ABB RAPID module: P701.mod

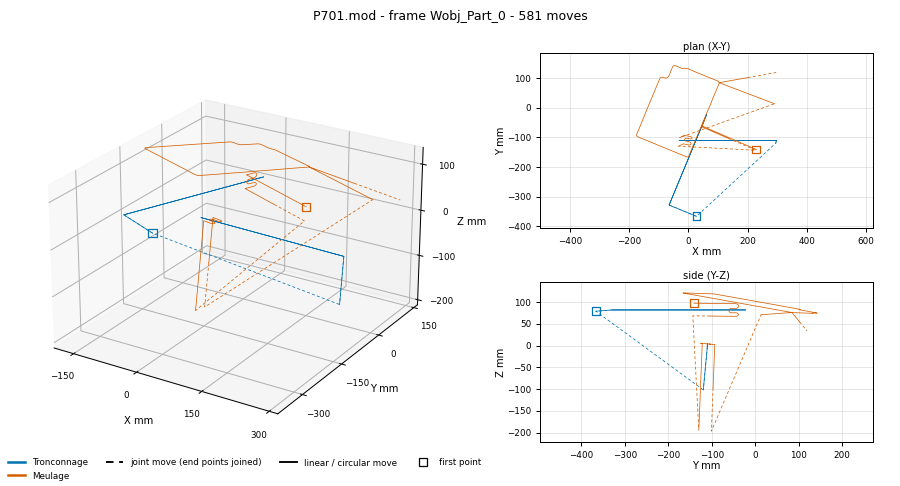
[picture p0: tool path of P701.mod in frame Wobj_Part_0, 581 of 591 moves have a stored position in this frame; points joined in program order, loops and branches not executed]
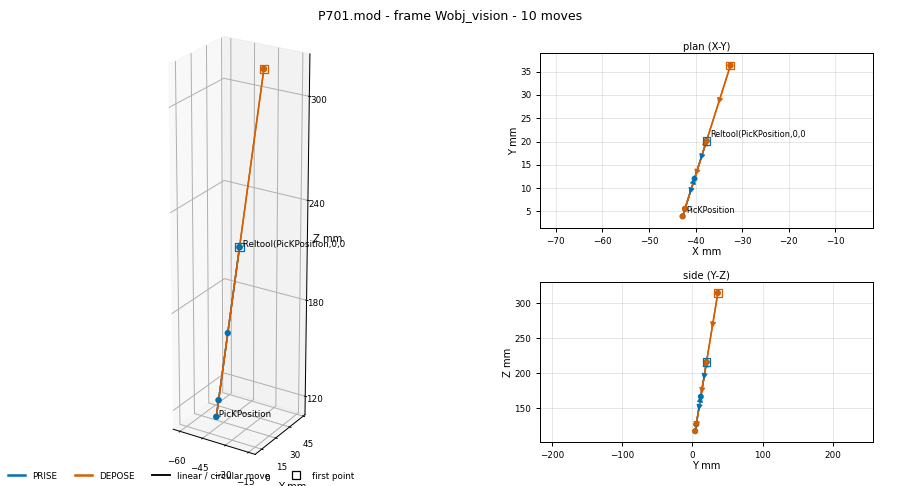
[picture p1: tool path of P701.mod in frame Wobj_vision, 10 of 591 moves have a stored position in this frame; points joined in program order, loops and branches not executed]
MODULE P701

    ! Nom         :P701
    ! Description :
    ! Créé le     :25/05/2023 17:26:44

    LOCAL CONST SPEEDDATA VitesseLente :=[10,500,0,0];
	LOCAL CONST SPEEDDATA VitesseRapide :=[30,500,0,0];
    !
    !Point de prise
    LOCAL PERS Robtarget PicKPosition := [[-42.7800235007069,3.94855808241573,117.453387874521],[0.0538335534292102,0.833835492186198,0.545408190576733,-0.0659562441896086],[0,0,0,0],[8.999999E+09,8.999999E+09,8.999999E+09,8.999999E+09,8.999999E+09,8.999999E+09]];
	LOCAL PERS Pose Ref := [[0,0,0],[1,0,0,0]];
    !
    !Declaration des points de meulage

    !Tr_meulage_motif_1 : Meulage d'un motif
    LOCAL CONST Robtarget Tr_meulage_motif_1_0 := [[45.67339453125,-61.43734375,96.697234375],[0.589642666457992,-0.592820387806933,-0.388910456451629,0.386825762527953],[0,0,0,0],[8.999999E+09,8.999999E+09,8.999999E+09,8.999999E+09,8.999999E+09,8.999999E+09]];
    LOCAL CONST Robtarget Tr_meulage_motif_1_1 := [[46.0576171875,-60.5141015625,96.6973125],[0.589642666457992,-0.592820387806933,-0.388910456451629,0.386825762527953],[0,0,0,0],[8.999999E+09,8.999999E+09,8.999999E+09,8.999999E+09,8.999999E+09,8.999999E+09]];
    LOCAL CONST Robtarget Tr_meulage_motif_1_2 := [[46.44183984375,-59.590859375,96.6973828125],[0.589642666457992,-0.592820387806933,-0.388910456451629,0.386825762527953],[0,0,0,0],[8.999999E+09,8.999999E+09,8.999999E+09,8.999999E+09,8.999999E+09,8.999999E+09]];
    LOCAL CONST Robtarget Tr_meulage_motif_1_3 := [[46.8260625,-58.66762109375,96.6974609375],[0.589642666457992,-0.592820387806933,-0.388910456451629,0.386825762527953],[0,0,0,0],[8.999999E+09,8.999999E+09,8.999999E+09,8.999999E+09,8.999999E+09,8.999999E+09]];
    LOCAL CONST Robtarget Tr_meulage_motif_1_4 := [[47.21028125,-57.74437890625,96.6975390625],[0.589642666457992,-0.592820387806933,-0.388910456451629,0.386825762527953],[0,0,0,0],[8.999999E+09,8.999999E+09,8.999999E+09,8.999999E+09,8.999999E+09,8.999999E+09]];
    LOCAL CONST Robtarget Tr_meulage_motif_1_5 := [[47.59450390625,-56.82113671875,96.697609375],[0.589642666457992,-0.592820387806933,-0.388910456451629,0.386825762527953],[0,0,0,0],[8.999999E+09,8.999999E+09,8.999999E+09,8.999999E+09,8.999999E+09,8.999999E+09]];
    LOCAL CONST Robtarget Tr_meulage_motif_1_6 := [[47.9787265625,-55.8978984375,96.6976875],[0.589642666457992,-0.592820387806933,-0.388910456451629,0.386825762527953],[0,0,0,0],[8.999999E+09,8.999999E+09,8.999999E+09,8.999999E+09,8.999999E+09,8.999999E+09]];
    LOCAL CONST Robtarget Tr_meulage_motif_1_7 := [[48.36294921875,-54.97465625,96.697765625],[0.589642666457992,-0.592820387806933,-0.388910456451629,0.386825762527953],[0,0,0,0],[8.999999E+09,8.999999E+09,8.999999E+09,8.999999E+09,8.999999E+09,8.999999E+09]];
    LOCAL CONST Robtarget Tr_meulage_motif_1_8 := [[48.74716796875,-54.0514140625,96.69784375],[0.589642666457992,-0.592820387806933,-0.388910456451629,0.386825762527953],[0,0,0,0],[8.999999E+09,8.999999E+09,8.999999E+09,8.999999E+09,8.999999E+09,8.999999E+09]];
    LOCAL CONST Robtarget Tr_meulage_motif_1_9 := [[49.131390625,-53.12817578125,96.6979140625],[0.589642666457992,-0.592820387806933,-0.388910456451629,0.386825762527953],[0,0,0,0],[8.999999E+09,8.999999E+09,8.999999E+09,8.999999E+09,8.999999E+09,8.999999E+09]];
    LOCAL CONST Robtarget Tr_meulage_motif_1_10 := [[49.51561328125,-52.20493359375,96.6979921875],[0.589642666457992,-0.592820387806933,-0.388910456451629,0.386825762527953],[0,0,0,0],[8.999999E+09,8.999999E+09,8.999999E+09,8.999999E+09,8.999999E+09,8.999999E+09]];
    LOCAL CONST Robtarget Tr_meulage_motif_1_11 := [[49.8998359375,-51.28169140625,96.6980703125],[0.589642666457992,-0.592820387806933,-0.388910456451629,0.386825762527953],[0,0,0,0],[8.999999E+09,8.999999E+09,8.999999E+09,8.999999E+09,8.999999E+09,8.999999E+09]];
    LOCAL CONST Robtarget Tr_meulage_motif_1_12 := [[50.28405859375,-50.358453125,96.698140625],[0.589642666457992,-0.592820387806933,-0.388910456451629,0.386825762527953],[0,0,0,0],[8.999999E+09,8.999999E+09,8.999999E+09,8.999999E+09,8.999999E+09,8.999999E+09]];
    LOCAL CONST Robtarget Tr_meulage_motif_1_13 := [[50.66827734375,-49.4352109375,96.69821875],[0.589642666457992,-0.592820387806933,-0.388910456451629,0.386825762527953],[0,0,0,0],[8.999999E+09,8.999999E+09,8.999999E+09,8.999999E+09,8.999999E+09,8.999999E+09]];
    LOCAL CONST Robtarget Tr_meulage_motif_1_14 := [[51.0525,-48.51196875,96.698296875],[0.589642666457992,-0.592820387806933,-0.388910456451629,0.386825762527953],[0,0,0,0],[8.999999E+09,8.999999E+09,8.999999E+09,8.999999E+09,8.999999E+09,8.999999E+09]];
    LOCAL CONST Robtarget Tr_meulage_motif_1_15 := [[51.43672265625,-47.58873046875,96.698375],[0.589642666457992,-0.592820387806933,-0.388910456451629,0.386825762527953],[0,0,0,0],[8.999999E+09,8.999999E+09,8.999999E+09,8.999999E+09,8.999999E+09,8.999999E+09]];
    LOCAL CONST Robtarget Tr_meulage_motif_1_16 := [[51.8209453125,-46.66548828125,96.6984453125],[0.589642666457992,-0.592820387806933,-0.388910456451629,0.386825762527953],[0,0,0,0],[8.999999E+09,8.999999E+09,8.999999E+09,8.999999E+09,8.999999E+09,8.999999E+09]];
    LOCAL CONST Robtarget Tr_meulage_motif_1_17 := [[52.2051640625,-45.74225,96.6985234375],[0.589642666457992,-0.592820387806933,-0.388910456451629,0.386825762527953],[0,0,0,0],[8.999999E+09,8.999999E+09,8.999999E+09,8.999999E+09,8.999999E+09,8.999999E+09]];
    LOCAL CONST Robtarget Tr_meulage_motif_1_18 := [[52.58938671875,-44.8190078125,96.6986015625],[0.589642666457992,-0.592820387806933,-0.388910456451629,0.386825762527953],[0,0,0,0],[8.999999E+09,8.999999E+09,8.999999E+09,8.999999E+09,8.999999E+09,8.999999E+09]];
    LOCAL CONST Robtarget Tr_meulage_motif_1_19 := [[52.96788671875,-43.9014296875,96.588125],[0.589642666457992,-0.592820387806933,-0.388910456451629,0.386825762527953],[0,0,0,0],[8.999999E+09,8.999999E+09,8.999999E+09,8.999999E+09,8.999999E+09,8.999999E+09]];
    LOCAL CONST Robtarget Tr_meulage_motif_1_20 := [[53.326078125,-43.0252890625,96.37709375],[0.589642666457992,-0.592820387806933,-0.388910456451629,0.386825762527953],[0,0,0,0],[8.999999E+09,8.999999E+09,8.999999E+09,8.999999E+09,8.999999E+09,8.999999E+09]];
    LOCAL CONST Robtarget Tr_meulage_motif_1_21 := [[53.6466640625,-42.2350703125,96.105421875],[0.589642666457992,-0.592820387806933,-0.388910456451629,0.386825762527953],[0,0,0,0],[8.999999E+09,8.999999E+09,8.999999E+09,8.999999E+09,8.999999E+09,8.999999E+09]];
    LOCAL CONST Robtarget Tr_meulage_motif_1_22 := [[53.92765625,-41.53969921875,95.8296484375],[0.589642666457992,-0.592820387806933,-0.388910456451629,0.386825762527953],[0,0,0,0],[8.999999E+09,8.999999E+09,8.999999E+09,8.999999E+09,8.999999E+09,8.999999E+09]];
    LOCAL CONST Robtarget Tr_meulage_motif_1_23 := [[54.3347421875,-40.51645703125,95.2138515625],[0.589642666457992,-0.592820387806933,-0.388910456451629,0.386825762527953],[0,0,0,0],[8.999999E+09,8.999999E+09,8.999999E+09,8.999999E+09,8.999999E+09,8.999999E+09]];
    LOCAL CONST Robtarget Tr_meulage_motif_1_24 := [[54.70616796875,-39.5619609375,94.366609375],[0.589642666457992,-0.592820387806933,-0.388910456451629,0.386825762527953],[0,0,0,0],[8.999999E+09,8.999999E+09,8.999999E+09,8.999999E+09,8.999999E+09,8.999999E+09]];
    LOCAL CONST Robtarget Tr_meulage_motif_1_25 := [[55.0053203125,-38.7682421875,93.343203125],[0.589642666457992,-0.592820387806933,-0.388910456451629,0.386825762527953],[0,0,0,0],[8.999999E+09,8.999999E+09,8.999999E+09,8.999999E+09,8.999999E+09,8.999999E+09]];
    LOCAL CONST Robtarget Tr_meulage_motif_1_26 := [[55.16394921875,-38.30542578125,92.2274921875],[0.589642666457992,-0.592820387806933,-0.388910456451629,0.386825762527953],[0,0,0,0],[8.999999E+09,8.999999E+09,8.999999E+09,8.999999E+09,8.999999E+09,8.999999E+09]];
    LOCAL CONST Robtarget Tr_meulage_motif_1_27 := [[55.1563125,-38.272875,91.531796875],[0.589642666457992,-0.592820387806933,-0.388910456451629,0.386825762527953],[0,0,0,0],[8.999999E+09,8.999999E+09,8.999999E+09,8.999999E+09,8.999999E+09,8.999999E+09]];
    LOCAL CONST Robtarget Tr_meulage_motif_1_28 := [[55.139171875,-38.26569140625,90.8708125],[0.589642666457992,-0.592820387806933,-0.388910456451629,0.386825762527953],[0,0,0,0],[8.999999E+09,8.999999E+09,8.999999E+09,8.999999E+09,8.999999E+09,8.999999E+09]];
    LOCAL CONST Robtarget Tr_meulage_motif_1_29 := [[55.10095703125,-38.30916796875,90.2099765625],[0.589642666457992,-0.592820387806933,-0.388910456451629,0.386825762527953],[0,0,0,0],[8.999999E+09,8.999999E+09,8.999999E+09,8.999999E+09,8.999999E+09,8.999999E+09]];
    LOCAL CONST Robtarget Tr_meulage_motif_1_30 := [[54.88097265625,-38.75716796875,89.108625],[0.589642666457992,-0.592820387806933,-0.388910456451629,0.386825762527953],[0,0,0,0],[8.999999E+09,8.999999E+09,8.999999E+09,8.999999E+09,8.999999E+09,8.999999E+09]];
    LOCAL CONST Robtarget Tr_meulage_motif_1_31 := [[54.52575,-39.5371015625,88.102328125],[0.589642666457992,-0.592820387806933,-0.388910456451629,0.386825762527953],[0,0,0,0],[8.999999E+09,8.999999E+09,8.999999E+09,8.999999E+09,8.999999E+09,8.999999E+09]];
    LOCAL CONST Robtarget Tr_meulage_motif_1_32 := [[54.1110546875,-40.47294140625,87.273703125],[0.589642666457992,-0.592820387806933,-0.388910456451629,0.386825762527953],[0,0,0,0],[8.999999E+09,8.999999E+09,8.999999E+09,8.999999E+09,8.999999E+09,8.999999E+09]];
    LOCAL CONST Robtarget Tr_meulage_motif_1_33 := [[53.83680078125,-41.10299609375,86.8780625],[0.589642666457992,-0.592820387806933,-0.388910456451629,0.386825762527953],[0,0,0,0],[8.999999E+09,8.999999E+09,8.999999E+09,8.999999E+09,8.999999E+09,8.999999E+09]];
    LOCAL CONST Robtarget Tr_meulage_motif_1_34 := [[53.37917578125,-42.166953125,86.3906328125],[0.589642666457992,-0.592820387806933,-0.388910456451629,0.386825762527953],[0,0,0,0],[8.999999E+09,8.999999E+09,8.999999E+09,8.999999E+09,8.999999E+09,8.999999E+09]];
    LOCAL CONST Robtarget Tr_meulage_motif_1_35 := [[53.04765234375,-42.94425,86.126578125],[0.589642666457992,-0.592820387806933,-0.388910456451629,0.386825762527953],[0,0,0,0],[8.999999E+09,8.999999E+09,8.999999E+09,8.999999E+09,8.999999E+09,8.999999E+09]];
    LOCAL CONST Robtarget Tr_meulage_motif_1_36 := [[52.6842578125,-43.80248828125,85.9221171875],[0.589642666457992,-0.592820387806933,-0.388910456451629,0.386825762527953],[0,0,0,0],[8.999999E+09,8.999999E+09,8.999999E+09,8.999999E+09,8.999999E+09,8.999999E+09]];
    LOCAL CONST Robtarget Tr_meulage_motif_1_37 := [[52.30430859375,-44.70752734375,85.8134921875],[0.589642666457992,-0.592820387806933,-0.388910456451629,0.386825762527953],[0,0,0,0],[8.999999E+09,8.999999E+09,8.999999E+09,8.999999E+09,8.999999E+09,8.999999E+09]];
    LOCAL CONST Robtarget Tr_meulage_motif_1_38 := [[51.920078125,-45.62269921875,85.7028671875],[0.589642666457992,-0.592820387806933,-0.388910456451629,0.386825762527953],[0,0,0,0],[8.999999E+09,8.999999E+09,8.999999E+09,8.999999E+09,8.999999E+09,8.999999E+09]];
    LOCAL CONST Robtarget Tr_meulage_motif_1_39 := [[51.53585546875,-46.54594140625,85.702796875],[0.589642666457992,-0.592820387806933,-0.388910456451629,0.386825762527953],[0,0,0,0],[8.999999E+09,8.999999E+09,8.999999E+09,8.999999E+09,8.999999E+09,8.999999E+09]];
    LOCAL CONST Robtarget Tr_meulage_motif_1_40 := [[51.1516328125,-47.4691796875,85.70271875],[0.589642666457992,-0.592820387806933,-0.388910456451629,0.386825762527953],[0,0,0,0],[8.999999E+09,8.999999E+09,8.999999E+09,8.999999E+09,8.999999E+09,8.999999E+09]];
    LOCAL CONST Robtarget Tr_meulage_motif_1_41 := [[50.76741015625,-48.392421875,85.702640625],[0.589642666457992,-0.592820387806933,-0.388910456451629,0.386825762527953],[0,0,0,0],[8.999999E+09,8.999999E+09,8.999999E+09,8.999999E+09,8.999999E+09,8.999999E+09]];
    LOCAL CONST Robtarget Tr_meulage_motif_1_42 := [[50.38319140625,-49.3156640625,85.7025625],[0.589642666457992,-0.592820387806933,-0.388910456451629,0.386825762527953],[0,0,0,0],[8.999999E+09,8.999999E+09,8.999999E+09,8.999999E+09,8.999999E+09,8.999999E+09]];
    LOCAL CONST Robtarget Tr_meulage_motif_1_43 := [[49.99896875,-50.23890234375,85.7024921875],[0.589642666457992,-0.592820387806933,-0.388910456451629,0.386825762527953],[0,0,0,0],[8.999999E+09,8.999999E+09,8.999999E+09,8.999999E+09,8.999999E+09,8.999999E+09]];
    LOCAL CONST Robtarget Tr_meulage_motif_1_44 := [[49.61474609375,-51.16214453125,85.7024140625],[0.589642666457992,-0.592820387806933,-0.388910456451629,0.386825762527953],[0,0,0,0],[8.999999E+09,8.999999E+09,8.999999E+09,8.999999E+09,8.999999E+09,8.999999E+09]];
    LOCAL CONST Robtarget Tr_meulage_motif_1_45 := [[49.2305234375,-52.08538671875,85.7023359375],[0.589642666457992,-0.592820387806933,-0.388910456451629,0.386825762527953],[0,0,0,0],[8.999999E+09,8.999999E+09,8.999999E+09,8.999999E+09,8.999999E+09,8.999999E+09]];
    LOCAL CONST Robtarget Tr_meulage_motif_1_46 := [[48.84630078125,-53.008625,85.7022578125],[0.589642666457992,-0.592820387806933,-0.388910456451629,0.386825762527953],[0,0,0,0],[8.999999E+09,8.999999E+09,8.999999E+09,8.999999E+09,8.999999E+09,8.999999E+09]];
    LOCAL CONST Robtarget Tr_meulage_motif_1_47 := [[48.46208203125,-53.9318671875,85.7021875],[0.589642666457992,-0.592820387806933,-0.388910456451629,0.386825762527953],[0,0,0,0],[8.999999E+09,8.999999E+09,8.999999E+09,8.999999E+09,8.999999E+09,8.999999E+09]];
    LOCAL CONST Robtarget Tr_meulage_motif_1_48 := [[48.077859375,-54.855109375,85.702109375],[0.589642666457992,-0.592820387806933,-0.388910456451629,0.386825762527953],[0,0,0,0],[8.999999E+09,8.999999E+09,8.999999E+09,8.999999E+09,8.999999E+09,8.999999E+09]];
    LOCAL CONST Robtarget Tr_meulage_motif_1_49 := [[47.69362890625,-55.77028125,85.591484375],[0.589642666457992,-0.592820387806933,-0.388910456451629,0.386825762527953],[0,0,0,0],[8.999999E+09,8.999999E+09,8.999999E+09,8.999999E+09,8.999999E+09,8.999999E+09]];
    LOCAL CONST Robtarget Tr_meulage_motif_1_50 := [[47.32448828125,-56.64183203125,85.3803046875],[0.589642666457992,-0.592820387806933,-0.388910456451629,0.386825762527953],[0,0,0,0],[8.999999E+09,8.999999E+09,8.999999E+09,8.999999E+09,8.999999E+09,8.999999E+09]];
    LOCAL CONST Robtarget Tr_meulage_motif_1_51 := [[46.98980859375,-57.426140625,85.1085078125],[0.589642666457992,-0.592820387806933,-0.388910456451629,0.386825762527953],[0,0,0,0],[8.999999E+09,8.999999E+09,8.999999E+09,8.999999E+09,8.999999E+09,8.999999E+09]];
    LOCAL CONST Robtarget Tr_meulage_motif_1_52 := [[46.7085546875,-58.07972265625,84.8044140625],[0.589642666457992,-0.592820387806933,-0.388910456451629,0.386825762527953],[0,0,0,0],[8.999999E+09,8.999999E+09,8.999999E+09,8.999999E+09,8.999999E+09,8.999999E+09]];
    LOCAL CONST Robtarget Tr_meulage_motif_1_53 := [[46.29391796875,-59.0275859375,84.1420703125],[0.589642666457992,-0.592820387806933,-0.388910456451629,0.386825762527953],[0,0,0,0],[8.999999E+09,8.999999E+09,8.999999E+09,8.999999E+09,8.999999E+09,8.999999E+09]];
    LOCAL CONST Robtarget Tr_meulage_motif_1_54 := [[45.92399609375,-59.85048828125,83.240421875],[0.589642666457992,-0.592820387806933,-0.388910456451629,0.386825762527953],[0,0,0,0],[8.999999E+09,8.999999E+09,8.999999E+09,8.999999E+09,8.999999E+09,8.999999E+09]];
    LOCAL CONST Robtarget Tr_meulage_motif_1_55 := [[45.69133984375,-60.33302734375,82.1947578125],[0.589642666457992,-0.592820387806933,-0.388910456451629,0.386825762527953],[0,0,0,0],[8.999999E+09,8.999999E+09,8.999999E+09,8.999999E+09,8.999999E+09,8.999999E+09]];
    LOCAL CONST Robtarget Tr_meulage_motif_1_56 := [[45.60237890625,-60.49608984375,81.5018046875],[0.589642666457992,-0.592820387806933,-0.388910456451629,0.386825762527953],[0,0,0,0],[8.999999E+09,8.999999E+09,8.999999E+09,8.999999E+09,8.999999E+09,8.999999E+09]];
    LOCAL CONST Robtarget Tr_meulage_motif_1_57 := [[45.557890625,-60.5466640625,80.7321015625],[0.589642666457992,-0.592820387806933,-0.388910456451629,0.386825762527953],[0,0,0,0],[8.999999E+09,8.999999E+09,8.999999E+09,8.999999E+09,8.999999E+09,8.999999E+09]];
    LOCAL CONST Robtarget Tr_meulage_motif_1_58 := [[45.56365625,-60.47649609375,79.96253125],[0.589642666457992,-0.592820387806933,-0.388910456451629,0.386825762527953],[0,0,0,0],[8.999999E+09,8.999999E+09,8.999999E+09,8.999999E+09,8.999999E+09,8.999999E+09]];
    LOCAL CONST Robtarget Tr_meulage_motif_1_59 := [[45.69615234375,-60.07706640625,78.8547578125],[0.589642666457992,-0.592820387806933,-0.388910456451629,0.386825762527953],[0,0,0,0],[8.999999E+09,8.999999E+09,8.999999E+09,8.999999E+09,8.999999E+09,8.999999E+09]];
    LOCAL CONST Robtarget Tr_meulage_motif_1_60 := [[45.84016015625,-59.68819140625,78.269328125],[0.589642666457992,-0.592820387806933,-0.388910456451629,0.386825762527953],[0,0,0,0],[8.999999E+09,8.999999E+09,8.999999E+09,8.999999E+09,8.999999E+09,8.999999E+09]];
    LOCAL CONST Robtarget Tr_meulage_motif_1_61 := [[46.15801953125,-58.85951953125,77.382625],[0.589642666457992,-0.592820387806933,-0.388910456451629,0.386825762527953],[0,0,0,0],[8.999999E+09,8.999999E+09,8.999999E+09,8.999999E+09,8.999999E+09,8.999999E+09]];
    LOCAL CONST Robtarget Tr_meulage_motif_1_62 := [[46.37231640625,-58.31428515625,76.968515625],[0.589642666457992,-0.592820387806933,-0.388910456451629,0.386825762527953],[0,0,0,0],[8.999999E+09,8.999999E+09,8.999999E+09,8.999999E+09,8.999999E+09,8.999999E+09]];
    LOCAL CONST Robtarget Tr_meulage_motif_1_63 := [[46.78773828125,-57.27627734375,76.4247265625],[0.589642666457992,-0.592820387806933,-0.388910456451629,0.386825762527953],[0,0,0,0],[8.999999E+09,8.999999E+09,8.999999E+09,8.999999E+09,8.999999E+09,8.999999E+09]];
    LOCAL CONST Robtarget Tr_meulage_motif_1_64 := [[47.09729296875,-56.51084375,76.12940625],[0.589642666457992,-0.592820387806933,-0.388910456451629,0.386825762527953],[0,0,0,0],[8.999999E+09,8.999999E+09,8.999999E+09,8.999999E+09,8.999999E+09,8.999999E+09]];
    LOCAL CONST Robtarget Tr_meulage_motif_1_65 := [[47.4500859375,-55.64816015625,75.9250859375],[0.589642666457992,-0.592820387806933,-0.388910456451629,0.386825762527953],[0,0,0,0],[8.999999E+09,8.999999E+09,8.999999E+09,8.999999E+09,8.999999E+09,8.999999E+09]];
    LOCAL CONST Robtarget Tr_meulage_motif_1_66 := [[47.82441015625,-54.74076171875,75.816609375],[0.589642666457992,-0.592820387806933,-0.388910456451629,0.386825762527953],[0,0,0,0],[8.999999E+09,8.999999E+09,8.999999E+09,8.999999E+09,8.999999E+09,8.999999E+09]];
    LOCAL CONST Robtarget Tr_meulage_motif_1_67 := [[48.20291015625,-53.8231875,75.7061328125],[0.589642666457992,-0.592820387806933,-0.388910456451629,0.386825762527953],[0,0,0,0],[8.999999E+09,8.999999E+09,8.999999E+09,8.999999E+09,8.999999E+09,8.999999E+09]];
    LOCAL CONST Robtarget Tr_meulage_motif_1_68 := [[48.58712890625,-52.8999453125,75.7062109375],[0.589642666457992,-0.592820387806933,-0.388910456451629,0.386825762527953],[0,0,0,0],[8.999999E+09,8.999999E+09,8.999999E+09,8.999999E+09,8.999999E+09,8.999999E+09]];
    LOCAL CONST Robtarget Tr_meulage_motif_1_69 := [[48.9713515625,-51.976703125,75.7062890625],[0.589642666457992,-0.592820387806933,-0.388910456451629,0.386825762527953],[0,0,0,0],[8.999999E+09,8.999999E+09,8.999999E+09,8.999999E+09,8.999999E+09,8.999999E+09]];
    LOCAL CONST Robtarget Tr_meulage_motif_1_70 := [[49.35557421875,-51.05346484375,75.706359375],[0.589642666457992,-0.592820387806933,-0.388910456451629,0.386825762527953],[0,0,0,0],[8.999999E+09,8.999999E+09,8.999999E+09,8.999999E+09,8.999999E+09,8.999999E+09]];
    LOCAL CONST Robtarget Tr_meulage_motif_1_71 := [[49.739796875,-50.13022265625,75.7064375],[0.589642666457992,-0.592820387806933,-0.388910456451629,0.386825762527953],[0,0,0,0],[8.999999E+09,8.999999E+09,8.999999E+09,8.999999E+09,8.999999E+09,8.999999E+09]];
    LOCAL CONST Robtarget Tr_meulage_motif_1_72 := [[50.12401953125,-49.20698046875,75.706515625],[0.589642666457992,-0.592820387806933,-0.388910456451629,0.386825762527953],[0,0,0,0],[8.999999E+09,8.999999E+09,8.999999E+09,8.999999E+09,8.999999E+09,8.999999E+09]];
    LOCAL CONST Robtarget Tr_meulage_motif_1_73 := [[50.50823828125,-48.2837421875,75.70659375],[0.589642666457992,-0.592820387806933,-0.388910456451629,0.386825762527953],[0,0,0,0],[8.999999E+09,8.999999E+09,8.999999E+09,8.999999E+09,8.999999E+09,8.999999E+09]];
    LOCAL CONST Robtarget Tr_meulage_motif_1_74 := [[50.8924609375,-47.3605,75.7066640625],[0.589642666457992,-0.592820387806933,-0.388910456451629,0.386825762527953],[0,0,0,0],[8.999999E+09,8.999999E+09,8.999999E+09,8.999999E+09,8.999999E+09,8.999999E+09]];
    LOCAL CONST Robtarget Tr_meulage_motif_1_75 := [[51.27668359375,-46.4372578125,75.7067421875],[0.589642666457992,-0.592820387806933,-0.388910456451629,0.386825762527953],[0,0,0,0],[8.999999E+09,8.999999E+09,8.999999E+09,8.999999E+09,8.999999E+09,8.999999E+09]];
    LOCAL CONST Robtarget Tr_meulage_motif_1_76 := [[51.66090625,-45.51401953125,75.7068203125],[0.589642666457992,-0.592820387806933,-0.388910456451629,0.386825762527953],[0,0,0,0],[8.999999E+09,8.999999E+09,8.999999E+09,8.999999E+09,8.999999E+09,8.999999E+09]];
    LOCAL CONST Robtarget Tr_meulage_motif_1_77 := [[52.045125,-44.59077734375,75.7068984375],[0.589642666457992,-0.592820387806933,-0.388910456451629,0.386825762527953],[0,0,0,0],[8.999999E+09,8.999999E+09,8.999999E+09,8.999999E+09,8.999999E+09,8.999999E+09]];
    LOCAL CONST Robtarget Tr_meulage_motif_1_78 := [[52.423625,-43.673203125,75.596421875],[0.589642666457992,-0.592820387806933,-0.388910456451629,0.386825762527953],[0,0,0,0],[8.999999E+09,8.999999E+09,8.999999E+09,8.999999E+09,8.999999E+09,8.999999E+09]];
    LOCAL CONST Robtarget Tr_meulage_motif_1_79 := [[52.78181640625,-42.79705859375,75.385390625],[0.589642666457992,-0.592820387806933,-0.388910456451629,0.386825762527953],[0,0,0,0],[8.999999E+09,8.999999E+09,8.999999E+09,8.999999E+09,8.999999E+09,8.999999E+09]];
    LOCAL CONST Robtarget Tr_meulage_motif_1_80 := [[53.10240625,-42.00683984375,75.11371875],[0.589642666457992,-0.592820387806933,-0.388910456451629,0.386825762527953],[0,0,0,0],[8.999999E+09,8.999999E+09,8.999999E+09,8.999999E+09,8.999999E+09,8.999999E+09]];
    LOCAL CONST Robtarget Tr_meulage_motif_1_81 := [[53.38339453125,-41.31146875,74.8379453125],[0.589642666457992,-0.592820387806933,-0.388910456451629,0.386825762527953],[0,0,0,0],[8.999999E+09,8.999999E+09,8.999999E+09,8.999999E+09,8.999999E+09,8.999999E+09]];
    LOCAL CONST Robtarget Tr_meulage_motif_1_82 := [[53.79048046875,-40.2882265625,74.2221484375],[0.589642666457992,-0.592820387806933,-0.388910456451629,0.386825762527953],[0,0,0,0],[8.999999E+09,8.999999E+09,8.999999E+09,8.999999E+09,8.999999E+09,8.999999E+09]];
    LOCAL CONST Robtarget Tr_meulage_motif_1_83 := [[54.13490234375,-39.39523046875,73.3286015625],[0.589642666457992,-0.592820387806933,-0.388910456451629,0.386825762527953],[0,0,0,0],[8.999999E+09,8.999999E+09,8.999999E+09,8.999999E+09,8.999999E+09,8.999999E+09]];
    LOCAL CONST Robtarget Tr_meulage_motif_1_84 := [[54.340796875,-38.82105859375,72.243078125],[0.589642666457992,-0.592820387806933,-0.388910456451629,0.386825762527953],[0,0,0,0],[8.999999E+09,8.999999E+09,8.999999E+09,8.999999E+09,8.999999E+09,8.999999E+09]];
    LOCAL CONST Robtarget Tr_meulage_motif_1_85 := [[54.3803359375,-38.65404296875,71.2591015625],[0.589642666457992,-0.592820387806933,-0.388910456451629,0.386825762527953],[0,0,0,0],[8.999999E+09,8.999999E+09,8.999999E+09,8.999999E+09,8.999999E+09,8.999999E+09]];
    LOCAL CONST Robtarget Tr_meulage_motif_1_86 := [[54.32451953125,-38.7731953125,71.0545234375],[0.589642666457992,-0.592820387806933,-0.388910456451629,0.386825762527953],[0,0,0,0],[8.999999E+09,8.999999E+09,8.999999E+09,8.999999E+09,8.999999E+09,8.999999E+09]];
    LOCAL CONST Robtarget Tr_meulage_motif_1_87 := [[54.2582890625,-38.87920703125,70.328390625],[0.589642666457992,-0.592820387806933,-0.388910456451629,0.386825762527953],[0,0,0,0],[8.999999E+09,8.999999E+09,8.999999E+09,8.999999E+09,8.999999E+09,8.999999E+09]];
    LOCAL CONST Robtarget Tr_meulage_motif_1_88 := [[53.97119921875,-39.50051953125,69.3918046875],[0.589642666457992,-0.592820387806933,-0.388910456451629,0.386825762527953],[0,0,0,0],[8.999999E+09,8.999999E+09,8.999999E+09,8.999999E+09,8.999999E+09,8.999999E+09]];
    LOCAL CONST Robtarget Tr_meulage_motif_1_89 := [[53.7449296875,-40.01030078125,68.9281328125],[0.589642666457992,-0.592820387806933,-0.388910456451629,0.386825762527953],[0,0,0,0],[8.999999E+09,8.999999E+09,8.999999E+09,8.999999E+09,8.999999E+09,8.999999E+09]];
    LOCAL CONST Robtarget Tr_meulage_motif_1_90 := [[53.296890625,-41.0480859375,68.3978203125],[0.589642666457992,-0.592820387806933,-0.388910456451629,0.386825762527953],[0,0,0,0],[8.999999E+09,8.999999E+09,8.999999E+09,8.999999E+09,8.999999E+09,8.999999E+09]];
    LOCAL CONST Robtarget Tr_meulage_motif_1_91 := [[52.9653671875,-41.8253828125,68.133765625],[0.589642666457992,-0.592820387806933,-0.388910456451629,0.386825762527953],[0,0,0,0],[8.999999E+09,8.999999E+09,8.999999E+09,8.999999E+09,8.999999E+09,8.999999E+09]];
    LOCAL CONST Robtarget Tr_meulage_motif_1_92 := [[52.60197265625,-42.68362109375,67.9293046875],[0.589642666457992,-0.592820387806933,-0.388910456451629,0.386825762527953],[0,0,0,0],[8.999999E+09,8.999999E+09,8.999999E+09,8.999999E+09,8.999999E+09,8.999999E+09]];
    LOCAL CONST Robtarget Tr_meulage_motif_1_93 := [[52.22201953125,-43.58866015625,67.8206796875],[0.589642666457992,-0.592820387806933,-0.388910456451629,0.386825762527953],[0,0,0,0],[8.999999E+09,8.999999E+09,8.999999E+09,8.999999E+09,8.999999E+09,8.999999E+09]];
    LOCAL CONST Robtarget Tr_meulage_motif_1_94 := [[51.8377890625,-44.50383203125,67.7100546875],[0.589642666457992,-0.592820387806933,-0.388910456451629,0.386825762527953],[0,0,0,0],[8.999999E+09,8.999999E+09,8.999999E+09,8.999999E+09,8.999999E+09,8.999999E+09]];
    LOCAL CONST Robtarget Tr_meulage_motif_1_95 := [[51.45356640625,-45.42707421875,67.7099765625],[0.589642666457992,-0.592820387806933,-0.388910456451629,0.386825762527953],[0,0,0,0],[8.999999E+09,8.999999E+09,8.999999E+09,8.999999E+09,8.999999E+09,8.999999E+09]];
    LOCAL CONST Robtarget Tr_meulage_motif_1_96 := [[51.06934765625,-46.35031640625,67.70990625],[0.589642666457992,-0.592820387806933,-0.388910456451629,0.386825762527953],[0,0,0,0],[8.999999E+09,8.999999E+09,8.999999E+09,8.999999E+09,8.999999E+09,8.999999E+09]];
    LOCAL CONST Robtarget Tr_meulage_motif_1_97 := [[50.685125,-47.2735546875,67.709828125],[0.589642666457992,-0.592820387806933,-0.388910456451629,0.386825762527953],[0,0,0,0],[8.999999E+09,8.999999E+09,8.999999E+09,8.999999E+09,8.999999E+09,8.999999E+09]];
    LOCAL CONST Robtarget Tr_meulage_motif_1_98 := [[50.30090234375,-48.196796875,67.70975],[0.589642666457992,-0.592820387806933,-0.388910456451629,0.386825762527953],[0,0,0,0],[8.999999E+09,8.999999E+09,8.999999E+09,8.999999E+09,8.999999E+09,8.999999E+09]];
    LOCAL CONST Robtarget Tr_meulage_motif_1_99 := [[49.9166796875,-49.1200390625,67.709671875],[0.589642666457992,-0.592820387806933,-0.388910456451629,0.386825762527953],[0,0,0,0],[8.999999E+09,8.999999E+09,8.999999E+09,8.999999E+09,8.999999E+09,8.999999E+09]];
    LOCAL CONST Robtarget Tr_meulage_motif_1_100 := [[49.53245703125,-50.04327734375,67.7096015625],[0.589642666457992,-0.592820387806933,-0.388910456451629,0.386825762527953],[0,0,0,0],[8.999999E+09,8.999999E+09,8.999999E+09,8.999999E+09,8.999999E+09,8.999999E+09]];
    LOCAL CONST Robtarget Tr_meulage_motif_1_101 := [[49.14823828125,-50.96651953125,67.7095234375],[0.589642666457992,-0.592820387806933,-0.388910456451629,0.386825762527953],[0,0,0,0],[8.999999E+09,8.999999E+09,8.999999E+09,8.999999E+09,8.999999E+09,8.999999E+09]];
    LOCAL CONST Robtarget Tr_meulage_motif_1_102 := [[48.764015625,-51.88976171875,67.7094453125],[0.589642666457992,-0.592820387806933,-0.388910456451629,0.386825762527953],[0,0,0,0],[8.999999E+09,8.999999E+09,8.999999E+09,8.999999E+09,8.999999E+09,8.999999E+09]];
    LOCAL CONST Robtarget Tr_meulage_motif_1_103 := [[48.37979296875,-52.813,67.709375],[0.589642666457992,-0.592820387806933,-0.388910456451629,0.386825762527953],[0,0,0,0],[8.999999E+09,8.999999E+09,8.999999E+09,8.999999E+09,8.999999E+09,8.999999E+09]];
    LOCAL CONST Robtarget Tr_meulage_motif_1_104 := [[47.9955703125,-53.7362421875,67.709296875],[0.589642666457992,-0.592820387806933,-0.388910456451629,0.386825762527953],[0,0,0,0],[8.999999E+09,8.999999E+09,8.999999E+09,8.999999E+09,8.999999E+09,8.999999E+09]];
    LOCAL CONST Robtarget Tr_meulage_motif_1_105 := [[47.6113515625,-54.65948046875,67.70921875],[0.589642666457992,-0.592820387806933,-0.388910456451629,0.386825762527953],[0,0,0,0],[8.999999E+09,8.999999E+09,8.999999E+09,8.999999E+09,8.999999E+09,8.999999E+09]];
    LOCAL CONST Robtarget Tr_meulage_motif_1_106 := [[47.22712890625,-55.58272265625,67.709140625],[0.589642666457992,-0.592820387806933,-0.388910456451629,0.386825762527953],[0,0,0,0],[8.999999E+09,8.999999E+09,8.999999E+09,8.999999E+09,8.999999E+09,8.999999E+09]];
    LOCAL CONST Robtarget Tr_meulage_motif_1_107 := [[46.84290625,-56.50596484375,67.7090703125],[0.589642666457992,-0.592820387806933,-0.388910456451629,0.386825762527953],[0,0,0,0],[8.999999E+09,8.999999E+09,8.999999E+09,8.999999E+09,8.999999E+09,8.999999E+09]];
    LOCAL CONST Robtarget Tr_meulage_motif_1_108 := [[46.45868359375,-57.429203125,67.7089921875],[0.589642666457992,-0.592820387806933,-0.388910456451629,0.386825762527953],[0,0,0,0],[8.999999E+09,8.999999E+09,8.999999E+09,8.999999E+09,8.999999E+09,8.999999E+09]];
    LOCAL CONST Robtarget Tr_meulage_motif_1_109 := [[46.0744609375,-58.3524453125,67.7089140625],[0.589642666457992,-0.592820387806933,-0.388910456451629,0.386825762527953],[0,0,0,0],[8.999999E+09,8.999999E+09,8.999999E+09,8.999999E+09,8.999999E+09,8.999999E+09]];
    LOCAL CONST Robtarget Tr_meulage_motif_1_110 := [[45.6902421875,-59.2756875,67.7088359375],[0.589642666457992,-0.592820387806933,-0.388910456451629,0.386825762527953],[0,0,0,0],[8.999999E+09,8.999999E+09,8.999999E+09,8.999999E+09,8.999999E+09,8.999999E+09]];
    LOCAL CONST Robtarget Tr_meulage_motif_1_111 := [[45.30601953125,-60.19892578125,67.708765625],[0.589642666457992,-0.592820387806933,-0.388910456451629,0.386825762527953],[0,0,0,0],[8.999999E+09,8.999999E+09,8.999999E+09,8.999999E+09,8.999999E+09,8.999999E+09]];
    LOCAL CONST Robtarget Tr_meulage_motif_1_112 := [[44.921796875,-61.12216796875,67.7086875],[0.589642666457992,-0.592820387806933,-0.388910456451629,0.386825762527953],[0,0,0,0],[8.999999E+09,8.999999E+09,8.999999E+09,8.999999E+09,8.999999E+09,8.999999E+09]];
    LOCAL CONST Robtarget Tr_meulage_motif_1_113 := [[44.53757421875,-62.04541015625,67.708609375],[0.589642666457992,-0.592820387806933,-0.388910456451629,0.386825762527953],[0,0,0,0],[8.999999E+09,8.999999E+09,8.999999E+09,8.999999E+09,8.999999E+09,8.999999E+09]];
    LOCAL CONST Robtarget Tr_meulage_motif_1_114 := [[44.15335546875,-62.9686484375,67.7085390625],[0.589642666457992,-0.592820387806933,-0.388910456451629,0.386825762527953],[0,0,0,0],[8.999999E+09,8.999999E+09,8.999999E+09,8.999999E+09,8.999999E+09,8.999999E+09]];
    LOCAL CONST Robtarget Tr_meulage_motif_1_115 := [[43.7691328125,-63.891890625,67.7084609375],[0.589642666457992,-0.592820387806933,-0.388910456451629,0.386825762527953],[0,0,0,0],[8.999999E+09,8.999999E+09,8.999999E+09,8.999999E+09,8.999999E+09,8.999999E+09]];

    !Tr_meulage_motif_2 : Meulage d'un motif
    LOCAL CONST Robtarget Tr_meulage_motif_2_0 := [[-17.13964453125,-121.794296875,5.3701357421875],[-0.000800740898031338,0.0405404313251403,0.0197315692809362,0.998982731290035],[0,0,0,0],[8.999999E+09,8.999999E+09,8.999999E+09,8.999999E+09,8.999999E+09,8.999999E+09]];
    LOCAL CONST Robtarget Tr_meulage_motif_2_1 := [[-16.1640869140625,-122.0132734375,5.38848095703125],[-0.000800740898031338,0.0405404313251403,0.0197315692809362,0.998982731290035],[0,0,0,0],[8.999999E+09,8.999999E+09,8.999999E+09,8.999999E+09,8.999999E+09,8.999999E+09]];
    LOCAL CONST Robtarget Tr_meulage_motif_2_2 := [[-15.188529296875,-122.23225,5.40682666015625],[-0.000800740898031338,0.0405404313251403,0.0197315692809362,0.998982731290035],[0,0,0,0],[8.999999E+09,8.999999E+09,8.999999E+09,8.999999E+09,8.999999E+09,8.999999E+09]];
    LOCAL CONST Robtarget Tr_meulage_motif_2_3 := [[-14.2129716796875,-122.4512265625,5.42517236328125],[-0.000800740898031338,0.0405404313251403,0.0197315692809362,0.998982731290035],[0,0,0,0],[8.999999E+09,8.999999E+09,8.999999E+09,8.999999E+09,8.999999E+09,8.999999E+09]];
    LOCAL CONST Robtarget Tr_meulage_motif_2_4 := [[-13.2374140625,-122.6702109375,5.44351806640625],[-0.000800740898031338,0.0405404313251403,0.0197315692809362,0.998982731290035],[0,0,0,0],[8.999999E+09,8.999999E+09,8.999999E+09,8.999999E+09,8.999999E+09,8.999999E+09]];
    LOCAL CONST Robtarget Tr_meulage_motif_2_5 := [[-12.2618564453125,-122.8891875,5.46186376953125],[-0.000800740898031338,0.0405404313251403,0.0197315692809362,0.998982731290035],[0,0,0,0],[8.999999E+09,8.999999E+09,8.999999E+09,8.999999E+09,8.999999E+09,8.999999E+09]];
    LOCAL CONST Robtarget Tr_meulage_motif_2_6 := [[-11.286298828125,-123.1081640625,5.48020947265625],[-0.000800740898031338,0.0405404313251403,0.0197315692809362,0.998982731290035],[0,0,0,0],[8.999999E+09,8.999999E+09,8.999999E+09,8.999999E+09,8.999999E+09,8.999999E+09]];
    LOCAL CONST Robtarget Tr_meulage_motif_2_7 := [[-10.3107412109375,-123.327140625,5.49855517578125],[-0.000800740898031338,0.0405404313251403,0.0197315692809362,0.998982731290035],[0,0,0,0],[8.999999E+09,8.999999E+09,8.999999E+09,8.999999E+09,8.999999E+09,8.999999E+09]];
    LOCAL CONST Robtarget Tr_meulage_motif_2_8 := [[-9.33518359375,-123.5461171875,5.516900390625],[-0.000800740898031338,0.0405404313251403,0.0197315692809362,0.998982731290035],[0,0,0,0],[8.999999E+09,8.999999E+09,8.999999E+09,8.999999E+09,8.999999E+09,8.999999E+09]];
    LOCAL CONST Robtarget Tr_meulage_motif_2_9 := [[-8.3596259765625,-123.76509375,5.53524609375],[-0.000800740898031338,0.0405404313251403,0.0197315692809362,0.998982731290035],[0,0,0,0],[8.999999E+09,8.999999E+09,8.999999E+09,8.999999E+09,8.999999E+09,8.999999E+09]];
    LOCAL CONST Robtarget Tr_meulage_motif_2_10 := [[-7.38406787109375,-123.9840703125,5.553591796875],[-0.000800740898031338,0.0405404313251403,0.0197315692809362,0.998982731290035],[0,0,0,0],[8.999999E+09,8.999999E+09,8.999999E+09,8.999999E+09,8.999999E+09,8.999999E+09]];
    LOCAL CONST Robtarget Tr_meulage_motif_2_11 := [[-6.40851025390625,-124.203046875,5.5719375],[-0.000800740898031338,0.0405404313251403,0.0197315692809362,0.998982731290035],[0,0,0,0],[8.999999E+09,8.999999E+09,8.999999E+09,8.999999E+09,8.999999E+09,8.999999E+09]];
    LOCAL CONST Robtarget Tr_meulage_motif_2_12 := [[-5.43295263671875,-124.4220234375,5.590283203125],[-0.000800740898031338,0.0405404313251403,0.0197315692809362,0.998982731290035],[0,0,0,0],[8.999999E+09,8.999999E+09,8.999999E+09,8.999999E+09,8.999999E+09,8.999999E+09]];
    LOCAL CONST Robtarget Tr_meulage_motif_2_13 := [[-4.45739501953125,-124.641,5.60862890625],[-0.000800740898031338,0.0405404313251403,0.0197315692809362,0.998982731290035],[0,0,0,0],[8.999999E+09,8.999999E+09,8.999999E+09,8.999999E+09,8.999999E+09,8.999999E+09]];
    LOCAL CONST Robtarget Tr_meulage_motif_2_14 := [[-3.48183764648437,-124.8599765625,5.62697412109375],[-0.000800740898031338,0.0405404313251403,0.0197315692809362,0.998982731290035],[0,0,0,0],[8.999999E+09,8.999999E+09,8.999999E+09,8.999999E+09,8.999999E+09,8.999999E+09]];
    LOCAL CONST Robtarget Tr_meulage_motif_2_15 := [[-2.50628002929687,-125.078953125,5.64531982421875],[-0.000800740898031338,0.0405404313251403,0.0197315692809362,0.998982731290035],[0,0,0,0],[8.999999E+09,8.999999E+09,8.999999E+09,8.999999E+09,8.999999E+09,8.999999E+09]];
    LOCAL CONST Robtarget Tr_meulage_motif_2_16 := [[-1.53072229003906,-125.2979296875,5.66366552734375],[-0.000800740898031338,0.0405404313251403,0.0197315692809362,0.998982731290035],[0,0,0,0],[8.999999E+09,8.999999E+09,8.999999E+09,8.999999E+09,8.999999E+09,8.999999E+09]];
    LOCAL CONST Robtarget Tr_meulage_motif_2_17 := [[-0.555164733886719,-125.51690625,5.68201123046875],[-0.000800740898031338,0.0405404313251403,0.0197315692809362,0.998982731290035],[0,0,0,0],[8.999999E+09,8.999999E+09,8.999999E+09,8.999999E+09,8.999999E+09,8.999999E+09]];
    LOCAL CONST Robtarget Tr_meulage_motif_2_18 := [[0.420392913818359,-125.7358828125,5.70035693359375],[-0.000800740898031338,0.0405404313251403,0.0197315692809362,0.998982731290035],[0,0,0,0],[8.999999E+09,8.999999E+09,8.999999E+09,8.999999E+09,8.999999E+09,8.999999E+09]];
    LOCAL CONST Robtarget Tr_meulage_motif_2_19 := [[1.41299609375,-125.845796875,5.7085703125],[-0.000800740898031338,0.0405404313251403,0.0197315692809362,0.998982731290035],[0,0,0,0],[8.999999E+09,8.999999E+09,8.999999E+09,8.999999E+09,8.999999E+09,8.999999E+09]];
    LOCAL CONST Robtarget Tr_meulage_motif_2_20 := [[2.3827666015625,-125.847921875,5.7068466796875],[-0.000800740898031338,0.0405404313251403,0.0197315692809362,0.998982731290035],[0,0,0,0],[8.999999E+09,8.999999E+09,8.999999E+09,8.999999E+09,8.999999E+09,8.999999E+09]];
    LOCAL CONST Robtarget Tr_meulage_motif_2_21 := [[3.27437646484375,-125.7705859375,5.697919921875],[-0.000800740898031338,0.0405404313251403,0.0197315692809362,0.998982731290035],[0,0,0,0],[8.999999E+09,8.999999E+09,8.999999E+09,8.999999E+09,8.999999E+09,8.999999E+09]];
    LOCAL CONST Robtarget Tr_meulage_motif_2_22 := [[4.06661694335938,-125.6667734375,5.68673779296875],[-0.000800740898031338,0.0405404313251403,0.0197315692809362,0.998982731290035],[0,0,0,0],[8.999999E+09,8.999999E+09,8.999999E+09,8.999999E+09,8.999999E+09,8.999999E+09]];
    LOCAL CONST Robtarget Tr_meulage_motif_2_23 := [[5.27615087890625,-125.3093984375,5.65125],[-0.000800740898031338,0.0405404313251403,0.0197315692809362,0.998982731290035],[0,0,0,0],[8.999999E+09,8.999999E+09,8.999999E+09,8.999999E+09,8.999999E+09,8.999999E+09]];
    LOCAL CONST Robtarget Tr_meulage_motif_2_24 := [[6.461259765625,-124.71021875,5.59341943359375],[-0.000800740898031338,0.0405404313251403,0.0197315692809362,0.998982731290035],[0,0,0,0],[8.999999E+09,8.999999E+09,8.999999E+09,8.999999E+09,8.999999E+09,8.999999E+09]];
    LOCAL CONST Robtarget Tr_meulage_motif_2_25 := [[7.51317822265625,-123.90128125,5.5164287109375],[-0.000800740898031338,0.0405404313251403,0.0197315692809362,0.998982731290035],[0,0,0,0],[8.999999E+09,8.999999E+09,8.999999E+09,8.999999E+09,8.999999E+09,8.999999E+09]];
    LOCAL CONST Robtarget Tr_meulage_motif_2_26 := [[8.23466796875,-122.923953125,5.4244990234375],[-0.000800740898031338,0.0405404313251403,0.0197315692809362,0.998982731290035],[0,0,0,0],[8.999999E+09,8.999999E+09,8.999999E+09,8.999999E+09,8.999999E+09,8.999999E+09]];
    LOCAL CONST Robtarget Tr_meulage_motif_2_27 := [[8.413998046875,-122.2538359375,5.36209130859375],[-0.000800740898031338,0.0405404313251403,0.0197315692809362,0.998982731290035],[0,0,0,0],[8.999999E+09,8.999999E+09,8.999999E+09,8.999999E+09,8.999999E+09,8.999999E+09]];
    LOCAL CONST Robtarget Tr_meulage_motif_2_28 := [[8.5592978515625,-121.6115234375,5.3023251953125],[-0.000800740898031338,0.0405404313251403,0.0197315692809362,0.998982731290035],[0,0,0,0],[8.999999E+09,8.999999E+09,8.999999E+09,8.999999E+09,8.999999E+09,8.999999E+09]];
    LOCAL CONST Robtarget Tr_meulage_motif_2_29 := [[8.651029296875,-120.95734375,5.24156640625],[-0.000800740898031338,0.0405404313251403,0.0197315692809362,0.998982731290035],[0,0,0,0],[8.999999E+09,8.999999E+09,8.999999E+09,8.999999E+09,8.999999E+09,8.999999E+09]];
    LOCAL CONST Robtarget Tr_meulage_motif_2_30 := [[8.4070810546875,-119.778046875,5.13284619140625],[-0.000800740898031338,0.0405404313251403,0.0197315692809362,0.998982731290035],[0,0,0,0],[8.999999E+09,8.999999E+09,8.999999E+09,8.999999E+09,8.999999E+09,8.999999E+09]];
    LOCAL CONST Robtarget Tr_meulage_motif_2_31 := [[7.79258447265625,-118.612671875,5.0261484375],[-0.000800740898031338,0.0405404313251403,0.0197315692809362,0.998982731290035],[0,0,0,0],[8.999999E+09,8.999999E+09,8.999999E+09,8.999999E+09,8.999999E+09,8.999999E+09]];
    LOCAL CONST Robtarget Tr_meulage_motif_2_32 := [[6.97632568359375,-117.5834296875,4.93245703125],[-0.000800740898031338,0.0405404313251403,0.0197315692809362,0.998982731290035],[0,0,0,0],[8.999999E+09,8.999999E+09,8.999999E+09,8.999999E+09,8.999999E+09,8.999999E+09]];
    LOCAL CONST Robtarget Tr_meulage_motif_2_33 := [[6.392986328125,-117.0485546875,4.88408251953125],[-0.000800740898031338,0.0405404313251403,0.0197315692809362,0.998982731290035],[0,0,0,0],[8.999999E+09,8.999999E+09,8.999999E+09,8.999999E+09,8.999999E+09,8.999999E+09]];
    LOCAL CONST Robtarget Tr_meulage_motif_2_34 := [[5.370265625,-116.321375,4.8187705078125],[-0.000800740898031338,0.0405404313251403,0.0197315692809362,0.998982731290035],[0,0,0,0],[8.999999E+09,8.999999E+09,8.999999E+09,8.999999E+09,8.999999E+09,8.999999E+09]];
    LOCAL CONST Robtarget Tr_meulage_motif_2_35 := [[4.60391943359375,-115.879796875,4.77939794921875],[-0.000800740898031338,0.0405404313251403,0.0197315692809362,0.998982731290035],[0,0,0,0],[8.999999E+09,8.999999E+09,8.999999E+09,8.999999E+09,8.999999E+09,8.999999E+09]];
    LOCAL CONST Robtarget Tr_meulage_motif_2_36 := [[3.73962890625,-115.4771015625,4.7438193359375],[-0.000800740898031338,0.0405404313251403,0.0197315692809362,0.998982731290035],[0,0,0,0],[8.999999E+09,8.999999E+09,8.999999E+09,8.999999E+09,8.999999E+09,8.999999E+09]];
    LOCAL CONST Robtarget Tr_meulage_motif_2_37 := [[2.805919921875,-115.1566796875,4.71599658203125],[-0.000800740898031338,0.0405404313251403,0.0197315692809362,0.998982731290035],[0,0,0,0],[8.999999E+09,8.999999E+09,8.999999E+09,8.999999E+09,8.999999E+09,8.999999E+09]];
    LOCAL CONST Robtarget Tr_meulage_motif_2_38 := [[1.86191931152344,-114.83190625,4.68779150390625],[-0.000800740898031338,0.0405404313251403,0.0197315692809362,0.998982731290035],[0,0,0,0],[8.999999E+09,8.999999E+09,8.999999E+09,8.999999E+09,8.999999E+09,8.999999E+09]];
    LOCAL CONST Robtarget Tr_meulage_motif_2_39 := [[0.886361633300781,-114.6129296875,4.6694462890625],[-0.000800740898031338,0.0405404313251403,0.0197315692809362,0.998982731290035],[0,0,0,0],[8.999999E+09,8.999999E+09,8.999999E+09,8.999999E+09,8.999999E+09,8.999999E+09]];
    LOCAL CONST Robtarget Tr_meulage_motif_2_40 := [[-0.0891959838867187,-114.393953125,4.6511005859375],[-0.000800740898031338,0.0405404313251403,0.0197315692809362,0.998982731290035],[0,0,0,0],[8.999999E+09,8.999999E+09,8.999999E+09,8.999999E+09,8.999999E+09,8.999999E+09]];
    LOCAL CONST Robtarget Tr_meulage_motif_2_41 := [[-1.06475366210937,-114.1749765625,4.6327548828125],[-0.000800740898031338,0.0405404313251403,0.0197315692809362,0.998982731290035],[0,0,0,0],[8.999999E+09,8.999999E+09,8.999999E+09,8.999999E+09,8.999999E+09,8.999999E+09]];
    LOCAL CONST Robtarget Tr_meulage_motif_2_42 := [[-2.04031127929687,-113.956,4.6144091796875],[-0.000800740898031338,0.0405404313251403,0.0197315692809362,0.998982731290035],[0,0,0,0],[8.999999E+09,8.999999E+09,8.999999E+09,8.999999E+09,8.999999E+09,8.999999E+09]];
    LOCAL CONST Robtarget Tr_meulage_motif_2_43 := [[-3.01586889648437,-113.7370234375,4.5960634765625],[-0.000800740898031338,0.0405404313251403,0.0197315692809362,0.998982731290035],[0,0,0,0],[8.999999E+09,8.999999E+09,8.999999E+09,8.999999E+09,8.999999E+09,8.999999E+09]];
    LOCAL CONST Robtarget Tr_meulage_motif_2_44 := [[-3.99142651367187,-113.5180390625,4.5777177734375],[-0.000800740898031338,0.0405404313251403,0.0197315692809362,0.998982731290035],[0,0,0,0],[8.999999E+09,8.999999E+09,8.999999E+09,8.999999E+09,8.999999E+09,8.999999E+09]];
    LOCAL CONST Robtarget Tr_meulage_motif_2_45 := [[-4.96698388671875,-113.2990625,4.55937255859375],[-0.000800740898031338,0.0405404313251403,0.0197315692809362,0.998982731290035],[0,0,0,0],[8.999999E+09,8.999999E+09,8.999999E+09,8.999999E+09,8.999999E+09,8.999999E+09]];
    LOCAL CONST Robtarget Tr_meulage_motif_2_46 := [[-5.94254150390625,-113.0800859375,4.54102685546875],[-0.000800740898031338,0.0405404313251403,0.0197315692809362,0.998982731290035],[0,0,0,0],[8.999999E+09,8.999999E+09,8.999999E+09,8.999999E+09,8.999999E+09,8.999999E+09]];
    LOCAL CONST Robtarget Tr_meulage_motif_2_47 := [[-6.918099609375,-112.861109375,4.52268115234375],[-0.000800740898031338,0.0405404313251403,0.0197315692809362,0.998982731290035],[0,0,0,0],[8.999999E+09,8.999999E+09,8.999999E+09,8.999999E+09,8.999999E+09,8.999999E+09]];
    LOCAL CONST Robtarget Tr_meulage_motif_2_48 := [[-7.8936572265625,-112.6421328125,4.50433544921875],[-0.000800740898031338,0.0405404313251403,0.0197315692809362,0.998982731290035],[0,0,0,0],[8.999999E+09,8.999999E+09,8.999999E+09,8.999999E+09,8.999999E+09,8.999999E+09]];
    LOCAL CONST Robtarget Tr_meulage_motif_2_49 := [[-8.8376572265625,-112.317359375,4.47613037109375],[-0.000800740898031338,0.0405404313251403,0.0197315692809362,0.998982731290035],[0,0,0,0],[8.999999E+09,8.999999E+09,8.999999E+09,8.999999E+09,8.999999E+09,8.999999E+09]];
    LOCAL CONST Robtarget Tr_meulage_motif_2_50 := [[-9.7146171875,-111.9049609375,4.43967822265625],[-0.000800740898031338,0.0405404313251403,0.0197315692809362,0.998982731290035],[0,0,0,0],[8.999999E+09,8.999999E+09,8.999999E+09,8.999999E+09,8.999999E+09,8.999999E+09]];
    LOCAL CONST Robtarget Tr_meulage_motif_2_51 := [[-10.4867607421875,-111.4541796875,4.39946435546875],[-0.000800740898031338,0.0405404313251403,0.0197315692809362,0.998982731290035],[0,0,0,0],[8.999999E+09,8.999999E+09,8.999999E+09,8.999999E+09,8.999999E+09,8.999999E+09]];
    LOCAL CONST Robtarget Tr_meulage_motif_2_52 := [[-11.1140361328125,-111.0029296875,4.3589208984375],[-0.000800740898031338,0.0405404313251403,0.0197315692809362,0.998982731290035],[0,0,0,0],[8.999999E+09,8.999999E+09,8.999999E+09,8.999999E+09,8.999999E+09,8.999999E+09]];
    LOCAL CONST Robtarget Tr_meulage_motif_2_53 := [[-11.977638671875,-110.13284375,4.28006103515625],[-0.000800740898031338,0.0405404313251403,0.0197315692809362,0.998982731290035],[0,0,0,0],[8.999999E+09,8.999999E+09,8.999999E+09,8.999999E+09,8.999999E+09,8.999999E+09]];
    LOCAL CONST Robtarget Tr_meulage_motif_2_54 := [[-12.65934375,-109.059234375,4.181994140625],[-0.000800740898031338,0.0405404313251403,0.0197315692809362,0.998982731290035],[0,0,0,0],[8.999999E+09,8.999999E+09,8.999999E+09,8.999999E+09,8.999999E+09,8.999999E+09]];
    LOCAL CONST Robtarget Tr_meulage_motif_2_55 := [[-12.95138671875,-107.9260078125,4.07763549804687],[-0.000800740898031338,0.0405404313251403,0.0197315692809362,0.998982731290035],[0,0,0,0],[8.999999E+09,8.999999E+09,8.999999E+09,8.999999E+09,8.999999E+09,8.999999E+09]];
    LOCAL CONST Robtarget Tr_meulage_motif_2_56 := [[-12.9793271484375,-107.2121796875,4.01159008789063],[-0.000800740898031338,0.0405404313251403,0.0197315692809362,0.998982731290035],[0,0,0,0],[8.999999E+09,8.999999E+09,8.999999E+09,8.999999E+09,8.999999E+09,8.999999E+09]];
    LOCAL CONST Robtarget Tr_meulage_motif_2_57 := [[-12.8724140625,-106.45025,3.94082348632813],[-0.000800740898031338,0.0405404313251403,0.0197315692809362,0.998982731290035],[0,0,0,0],[8.999999E+09,8.999999E+09,8.999999E+09,8.999999E+09,8.999999E+09,8.999999E+09]];
    LOCAL CONST Robtarget Tr_meulage_motif_2_58 := [[-12.6379443359375,-105.717078125,3.87246728515625],[-0.000800740898031338,0.0405404313251403,0.0197315692809362,0.998982731290035],[0,0,0,0],[8.999999E+09,8.999999E+09,8.999999E+09,8.999999E+09,8.999999E+09,8.999999E+09]];
    LOCAL CONST Robtarget Tr_meulage_motif_2_59 := [[-11.9850859375,-104.7324453125,3.77999755859375],[-0.000800740898031338,0.0405404313251403,0.0197315692809362,0.998982731290035],[0,0,0,0],[8.999999E+09,8.999999E+09,8.999999E+09,8.999999E+09,8.999999E+09,8.999999E+09]];
    LOCAL CONST Robtarget Tr_meulage_motif_2_60 := [[-11.4522041015625,-104.2542578125,3.73466162109375],[-0.000800740898031338,0.0405404313251403,0.0197315692809362,0.998982731290035],[0,0,0,0],[8.999999E+09,8.999999E+09,8.999999E+09,8.999999E+09,8.999999E+09,8.999999E+09]];
    LOCAL CONST Robtarget Tr_meulage_motif_2_61 := [[-10.391830078125,-103.586796875,3.67075512695313],[-0.000800740898031338,0.0405404313251403,0.0197315692809362,0.998982731290035],[0,0,0,0],[8.999999E+09,8.999999E+09,8.999999E+09,8.999999E+09,8.999999E+09,8.999999E+09]];
    LOCAL CONST Robtarget Tr_meulage_motif_2_62 := [[-9.7294189453125,-103.31259375,3.644052734375],[-0.000800740898031338,0.0405404313251403,0.0197315692809362,0.998982731290035],[0,0,0,0],[8.999999E+09,8.999999E+09,8.999999E+09,8.999999E+09,8.999999E+09,8.999999E+09]];
    LOCAL CONST Robtarget Tr_meulage_motif_2_63 := [[-8.5192802734375,-103.0288828125,3.61538427734375],[-0.000800740898031338,0.0405404313251403,0.0197315692809362,0.998982731290035],[0,0,0,0],[8.999999E+09,8.999999E+09,8.999999E+09,8.999999E+09,8.999999E+09,8.999999E+09]];
    LOCAL CONST Robtarget Tr_meulage_motif_2_64 := [[-7.6489345703125,-102.922625,3.60382202148438],[-0.000800740898031338,0.0405404313251403,0.0197315692809362,0.998982731290035],[0,0,0,0],[8.999999E+09,8.999999E+09,8.999999E+09,8.999999E+09,8.999999E+09,8.999999E+09]];
    LOCAL CONST Robtarget Tr_meulage_motif_2_65 := [[-6.6947861328125,-102.9281015625,3.602439453125],[-0.000800740898031338,0.0405404313251403,0.0197315692809362,0.998982731290035],[0,0,0,0],[8.999999E+09,8.999999E+09,8.999999E+09,8.999999E+09,8.999999E+09,8.999999E+09]];
    LOCAL CONST Robtarget Tr_meulage_motif_2_66 := [[-5.713353515625,-103.0375546875,3.6106318359375],[-0.000800740898031338,0.0405404313251403,0.0197315692809362,0.998982731290035],[0,0,0,0],[8.999999E+09,8.999999E+09,8.999999E+09,8.999999E+09,8.999999E+09,8.999999E+09]];
    LOCAL CONST Robtarget Tr_meulage_motif_2_67 := [[-4.72075048828125,-103.1474765625,3.61884521484375],[-0.000800740898031338,0.0405404313251403,0.0197315692809362,0.998982731290035],[0,0,0,0],[8.999999E+09,8.999999E+09,8.999999E+09,8.999999E+09,8.999999E+09,8.999999E+09]];
    LOCAL CONST Robtarget Tr_meulage_motif_2_68 := [[-3.74519262695313,-103.366453125,3.63719067382813],[-0.000800740898031338,0.0405404313251403,0.0197315692809362,0.998982731290035],[0,0,0,0],[8.999999E+09,8.999999E+09,8.999999E+09,8.999999E+09,8.999999E+09,8.999999E+09]];
    LOCAL CONST Robtarget Tr_meulage_motif_2_69 := [[-2.76963500976563,-103.5854296875,3.65553637695313],[-0.000800740898031338,0.0405404313251403,0.0197315692809362,0.998982731290035],[0,0,0,0],[8.999999E+09,8.999999E+09,8.999999E+09,8.999999E+09,8.999999E+09,8.999999E+09]];
    LOCAL CONST Robtarget Tr_meulage_motif_2_70 := [[-1.79407739257813,-103.80440625,3.67388208007812],[-0.000800740898031338,0.0405404313251403,0.0197315692809362,0.998982731290035],[0,0,0,0],[8.999999E+09,8.999999E+09,8.999999E+09,8.999999E+09,8.999999E+09,8.999999E+09]];
    LOCAL CONST Robtarget Tr_meulage_motif_2_71 := [[-0.818519775390625,-104.0233828125,3.69222778320312],[-0.000800740898031338,0.0405404313251403,0.0197315692809362,0.998982731290035],[0,0,0,0],[8.999999E+09,8.999999E+09,8.999999E+09,8.999999E+09,8.999999E+09,8.999999E+09]];
    LOCAL CONST Robtarget Tr_meulage_motif_2_72 := [[0.157037826538086,-104.242359375,3.7105732421875],[-0.000800740898031338,0.0405404313251403,0.0197315692809362,0.998982731290035],[0,0,0,0],[8.999999E+09,8.999999E+09,8.999999E+09,8.999999E+09,8.999999E+09,8.999999E+09]];
    LOCAL CONST Robtarget Tr_meulage_motif_2_73 := [[1.13259545898437,-104.4613359375,3.7289189453125],[-0.000800740898031338,0.0405404313251403,0.0197315692809362,0.998982731290035],[0,0,0,0],[8.999999E+09,8.999999E+09,8.999999E+09,8.999999E+09,8.999999E+09,8.999999E+09]];
    LOCAL CONST Robtarget Tr_meulage_motif_2_74 := [[2.10815307617188,-104.6803125,3.7472646484375],[-0.000800740898031338,0.0405404313251403,0.0197315692809362,0.998982731290035],[0,0,0,0],[8.999999E+09,8.999999E+09,8.999999E+09,8.999999E+09,8.999999E+09,8.999999E+09]];
    LOCAL CONST Robtarget Tr_meulage_motif_2_75 := [[3.08371069335938,-104.8992890625,3.76561010742188],[-0.000800740898031338,0.0405404313251403,0.0197315692809362,0.998982731290035],[0,0,0,0],[8.999999E+09,8.999999E+09,8.999999E+09,8.999999E+09,8.999999E+09,8.999999E+09]];
    LOCAL CONST Robtarget Tr_meulage_motif_2_76 := [[4.05926831054687,-105.118265625,3.78395581054688],[-0.000800740898031338,0.0405404313251403,0.0197315692809362,0.998982731290035],[0,0,0,0],[8.999999E+09,8.999999E+09,8.999999E+09,8.999999E+09,8.999999E+09,8.999999E+09]];
    LOCAL CONST Robtarget Tr_meulage_motif_2_77 := [[5.034826171875,-105.3372421875,3.80230151367188],[-0.000800740898031338,0.0405404313251403,0.0197315692809362,0.998982731290035],[0,0,0,0],[8.999999E+09,8.999999E+09,8.999999E+09,8.999999E+09,8.999999E+09,8.999999E+09]];
    LOCAL CONST Robtarget Tr_meulage_motif_2_78 := [[6.02742919921875,-105.4471640625,3.81051489257813],[-0.000800740898031338,0.0405404313251403,0.0197315692809362,0.998982731290035],[0,0,0,0],[8.999999E+09,8.999999E+09,8.999999E+09,8.999999E+09,8.999999E+09,8.999999E+09]];
    LOCAL CONST Robtarget Tr_meulage_motif_2_79 := [[6.99719970703125,-105.4492890625,3.808791015625],[-0.000800740898031338,0.0405404313251403,0.0197315692809362,0.998982731290035],[0,0,0,0],[8.999999E+09,8.999999E+09,8.999999E+09,8.999999E+09,8.999999E+09,8.999999E+09]];
    LOCAL CONST Robtarget Tr_meulage_motif_2_80 := [[7.8888095703125,-105.371953125,3.79986450195313],[-0.000800740898031338,0.0405404313251403,0.0197315692809362,0.998982731290035],[0,0,0,0],[8.999999E+09,8.999999E+09,8.999999E+09,8.999999E+09,8.999999E+09,8.999999E+09]];
    LOCAL CONST Robtarget Tr_meulage_motif_2_81 := [[8.6810498046875,-105.2681328125,3.78868237304688],[-0.000800740898031338,0.0405404313251403,0.0197315692809362,0.998982731290035],[0,0,0,0],[8.999999E+09,8.999999E+09,8.999999E+09,8.999999E+09,8.999999E+09,8.999999E+09]];
    LOCAL CONST Robtarget Tr_meulage_motif_2_82 := [[9.890583984375,-104.9107578125,3.7531943359375],[-0.000800740898031338,0.0405404313251403,0.0197315692809362,0.998982731290035],[0,0,0,0],[8.999999E+09,8.999999E+09,8.999999E+09,8.999999E+09,8.999999E+09,8.999999E+09]];
    LOCAL CONST Robtarget Tr_meulage_motif_2_83 := [[11.0203544921875,-104.251890625,3.68994604492188],[-0.000800740898031338,0.0405404313251403,0.0197315692809362,0.998982731290035],[0,0,0,0],[8.999999E+09,8.999999E+09,8.999999E+09,8.999999E+09,8.999999E+09,8.999999E+09]];
    LOCAL CONST Robtarget Tr_meulage_motif_2_84 := [[11.85322265625,-103.330375,3.60296411132812],[-0.000800740898031338,0.0405404313251403,0.0197315692809362,0.998982731290035],[0,0,0,0],[8.999999E+09,8.999999E+09,8.999999E+09,8.999999E+09,8.999999E+09,8.999999E+09]];
    LOCAL CONST Robtarget Tr_meulage_motif_2_85 := [[12.23469921875,-102.411265625,3.51709887695313],[-0.000800740898031338,0.0405404313251403,0.0197315692809362,0.998982731290035],[0,0,0,0],[8.999999E+09,8.999999E+09,8.999999E+09,8.999999E+09,8.999999E+09,8.999999E+09]];
    LOCAL CONST Robtarget Tr_meulage_motif_2_86 := [[12.1514130859375,-102.1836796875,3.496189453125],[-0.000800740898031338,0.0405404313251403,0.0197315692809362,0.998982731290035],[0,0,0,0],[8.999999E+09,8.999999E+09,8.999999E+09,8.999999E+09,8.999999E+09,8.999999E+09]];
    LOCAL CONST Robtarget Tr_meulage_motif_2_87 := [[12.1906708984375,-101.4510546875,3.42827099609375],[-0.000800740898031338,0.0405404313251403,0.0197315692809362,0.998982731290035],[0,0,0,0],[8.999999E+09,8.999999E+09,8.999999E+09,8.999999E+09,8.999999E+09,8.999999E+09]];
    LOCAL CONST Robtarget Tr_meulage_motif_2_88 := [[11.7292607421875,-100.391203125,3.33104150390625],[-0.000800740898031338,0.0405404313251403,0.0197315692809362,0.998982731290035],[0,0,0,0],[8.999999E+09,8.999999E+09,8.999999E+09,8.999999E+09,8.999999E+09,8.999999E+09]];
    LOCAL CONST Robtarget Tr_meulage_motif_2_89 := [[11.2871806640625,-99.8185625,3.278890625],[-0.000800740898031338,0.0405404313251403,0.0197315692809362,0.998982731290035],[0,0,0,0],[8.999999E+09,8.999999E+09,8.999999E+09,8.999999E+09,8.999999E+09,8.999999E+09]];
    LOCAL CONST Robtarget Tr_meulage_motif_2_90 := [[10.3010517578125,-99.0558046875,3.21021142578125],[-0.000800740898031338,0.0405404313251403,0.0197315692809362,0.998982731290035],[0,0,0,0],[8.999999E+09,8.999999E+09,8.999999E+09,8.999999E+09,8.999999E+09,8.999999E+09]];
    LOCAL CONST Robtarget Tr_meulage_motif_2_91 := [[9.534705078125,-98.614234375,3.17083911132812],[-0.000800740898031338,0.0405404313251403,0.0197315692809362,0.998982731290035],[0,0,0,0],[8.999999E+09,8.999999E+09,8.999999E+09,8.999999E+09,8.999999E+09,8.999999E+09]];
    LOCAL CONST Robtarget Tr_meulage_motif_2_92 := [[8.6704150390625,-98.21153125,3.13526025390625],[-0.000800740898031338,0.0405404313251403,0.0197315692809362,0.998982731290035],[0,0,0,0],[8.999999E+09,8.999999E+09,8.999999E+09,8.999999E+09,8.999999E+09,8.999999E+09]];
    LOCAL CONST Robtarget Tr_meulage_motif_2_93 := [[7.7367060546875,-97.891109375,3.10743774414063],[-0.000800740898031338,0.0405404313251403,0.0197315692809362,0.998982731290035],[0,0,0,0],[8.999999E+09,8.999999E+09,8.999999E+09,8.999999E+09,8.999999E+09,8.999999E+09]];
    LOCAL CONST Robtarget Tr_meulage_motif_2_94 := [[6.792705078125,-97.5663359375,3.07923266601563],[-0.000800740898031338,0.0405404313251403,0.0197315692809362,0.998982731290035],[0,0,0,0],[8.999999E+09,8.999999E+09,8.999999E+09,8.999999E+09,8.999999E+09,8.999999E+09]];
    LOCAL CONST Robtarget Tr_meulage_motif_2_95 := [[5.8171474609375,-97.347359375,3.06088720703125],[-0.000800740898031338,0.0405404313251403,0.0197315692809362,0.998982731290035],[0,0,0,0],[8.999999E+09,8.999999E+09,8.999999E+09,8.999999E+09,8.999999E+09,8.999999E+09]];
    LOCAL CONST Robtarget Tr_meulage_motif_2_96 := [[4.84158984375,-97.1283828125,3.04254150390625],[-0.000800740898031338,0.0405404313251403,0.0197315692809362,0.998982731290035],[0,0,0,0],[8.999999E+09,8.999999E+09,8.999999E+09,8.999999E+09,8.999999E+09,8.999999E+09]];
    LOCAL CONST Robtarget Tr_meulage_motif_2_97 := [[3.8660322265625,-96.90940625,3.02419580078125],[-0.000800740898031338,0.0405404313251403,0.0197315692809362,0.998982731290035],[0,0,0,0],[8.999999E+09,8.999999E+09,8.999999E+09,8.999999E+09,8.999999E+09,8.999999E+09]];
    LOCAL CONST Robtarget Tr_meulage_motif_2_98 := [[2.890474609375,-96.6904296875,3.00585009765625],[-0.000800740898031338,0.0405404313251403,0.0197315692809362,0.998982731290035],[0,0,0,0],[8.999999E+09,8.999999E+09,8.999999E+09,8.999999E+09,8.999999E+09,8.999999E+09]];
    LOCAL CONST Robtarget Tr_meulage_motif_2_99 := [[1.91491711425781,-96.471453125,2.98750463867187],[-0.000800740898031338,0.0405404313251403,0.0197315692809362,0.998982731290035],[0,0,0,0],[8.999999E+09,8.999999E+09,8.999999E+09,8.999999E+09,8.999999E+09,8.999999E+09]];
    LOCAL CONST Robtarget Tr_meulage_motif_2_100 := [[0.939359436035156,-96.2524765625,2.96915893554688],[-0.000800740898031338,0.0405404313251403,0.0197315692809362,0.998982731290035],[0,0,0,0],[8.999999E+09,8.999999E+09,8.999999E+09,8.999999E+09,8.999999E+09,8.999999E+09]];
    LOCAL CONST Robtarget Tr_meulage_motif_2_101 := [[-0.036198169708252,-96.0335,2.95081323242188],[-0.000800740898031338,0.0405404313251403,0.0197315692809362,0.998982731290035],[0,0,0,0],[8.999999E+09,8.999999E+09,8.999999E+09,8.999999E+09,8.999999E+09,8.999999E+09]];
    LOCAL CONST Robtarget Tr_meulage_motif_2_102 := [[-1.01175579833984,-95.8145234375,2.9324677734375],[-0.000800740898031338,0.0405404313251403,0.0197315692809362,0.998982731290035],[0,0,0,0],[8.999999E+09,8.999999E+09,8.999999E+09,8.999999E+09,8.999999E+09,8.999999E+09]];
    LOCAL CONST Robtarget Tr_meulage_motif_2_103 := [[-1.9873134765625,-95.595546875,2.9141220703125],[-0.000800740898031338,0.0405404313251403,0.0197315692809362,0.998982731290035],[0,0,0,0],[8.999999E+09,8.999999E+09,8.999999E+09,8.999999E+09,8.999999E+09,8.999999E+09]];
    LOCAL CONST Robtarget Tr_meulage_motif_2_104 := [[-2.96287109375,-95.3765703125,2.8957763671875],[-0.000800740898031338,0.0405404313251403,0.0197315692809362,0.998982731290035],[0,0,0,0],[8.999999E+09,8.999999E+09,8.999999E+09,8.999999E+09,8.999999E+09,8.999999E+09]];
    LOCAL CONST Robtarget Tr_meulage_motif_2_105 := [[-3.9384287109375,-95.15759375,2.87743090820313],[-0.000800740898031338,0.0405404313251403,0.0197315692809362,0.998982731290035],[0,0,0,0],[8.999999E+09,8.999999E+09,8.999999E+09,8.999999E+09,8.999999E+09,8.999999E+09]];
    LOCAL CONST Robtarget Tr_meulage_motif_2_106 := [[-4.913986328125,-94.9386171875,2.85908520507813],[-0.000800740898031338,0.0405404313251403,0.0197315692809362,0.998982731290035],[0,0,0,0],[8.999999E+09,8.999999E+09,8.999999E+09,8.999999E+09,8.999999E+09,8.999999E+09]];
    LOCAL CONST Robtarget Tr_meulage_motif_2_107 := [[-5.8895439453125,-94.719640625,2.84073950195312],[-0.000800740898031338,0.0405404313251403,0.0197315692809362,0.998982731290035],[0,0,0,0],[8.999999E+09,8.999999E+09,8.999999E+09,8.999999E+09,8.999999E+09,8.999999E+09]];
    LOCAL CONST Robtarget Tr_meulage_motif_2_108 := [[-6.8651015625,-94.5006640625,2.82239379882812],[-0.000800740898031338,0.0405404313251403,0.0197315692809362,0.998982731290035],[0,0,0,0],[8.999999E+09,8.999999E+09,8.999999E+09,8.999999E+09,8.999999E+09,8.999999E+09]];
    LOCAL CONST Robtarget Tr_meulage_motif_2_109 := [[-7.8406591796875,-94.2816875,2.80404833984375],[-0.000800740898031338,0.0405404313251403,0.0197315692809362,0.998982731290035],[0,0,0,0],[8.999999E+09,8.999999E+09,8.999999E+09,8.999999E+09,8.999999E+09,8.999999E+09]];
    LOCAL CONST Robtarget Tr_meulage_motif_2_110 := [[-8.816216796875,-94.0627109375,2.78570263671875],[-0.000800740898031338,0.0405404313251403,0.0197315692809362,0.998982731290035],[0,0,0,0],[8.999999E+09,8.999999E+09,8.999999E+09,8.999999E+09,8.999999E+09,8.999999E+09]];
    LOCAL CONST Robtarget Tr_meulage_motif_2_111 := [[-9.7917744140625,-93.843734375,2.76735693359375],[-0.000800740898031338,0.0405404313251403,0.0197315692809362,0.998982731290035],[0,0,0,0],[8.999999E+09,8.999999E+09,8.999999E+09,8.999999E+09,8.999999E+09,8.999999E+09]];
    LOCAL CONST Robtarget Tr_meulage_motif_2_112 := [[-10.76733203125,-93.6247578125,2.74901147460938],[-0.000800740898031338,0.0405404313251403,0.0197315692809362,0.998982731290035],[0,0,0,0],[8.999999E+09,8.999999E+09,8.999999E+09,8.999999E+09,8.999999E+09,8.999999E+09]];
    LOCAL CONST Robtarget Tr_meulage_motif_2_113 := [[-11.7428896484375,-93.40578125,2.73066577148438],[-0.000800740898031338,0.0405404313251403,0.0197315692809362,0.998982731290035],[0,0,0,0],[8.999999E+09,8.999999E+09,8.999999E+09,8.999999E+09,8.999999E+09,8.999999E+09]];
    LOCAL CONST Robtarget Tr_meulage_motif_2_114 := [[-12.718447265625,-93.1868046875,2.71232006835938],[-0.000800740898031338,0.0405404313251403,0.0197315692809362,0.998982731290035],[0,0,0,0],[8.999999E+09,8.999999E+09,8.999999E+09,8.999999E+09,8.999999E+09,8.999999E+09]];
    LOCAL CONST Robtarget Tr_meulage_motif_2_115 := [[-13.6940048828125,-92.967828125,2.693974609375],[-0.000800740898031338,0.0405404313251403,0.0197315692809362,0.998982731290035],[0,0,0,0],[8.999999E+09,8.999999E+09,8.999999E+09,8.999999E+09,8.999999E+09,8.999999E+09]];

